// TIA Portal V18 export
TYPE "TM_Pulse_2x24_In_PWM"
   STRUCT
      ERR_PWR : Bool;
      ERR_24V : Bool;
      ERR_LD : Bool;
      Reserved5 : Bool;
      ERR_DQA : Bool;
      ERR_DQB : Bool;
      ERR_OUT_VAL : Bool;
      ERR_SLOT_VAL : Bool;
      Reserved0 : Bool;
      Reserved1 : Bool;
      STS_LD_SLOT : Bool;
      Reserved2 : Bool;
      STS_READY : Bool;
      STS_SW_ENABLE : Bool;
      Reserved3 : Bool;
      Reserved4 : Bool;
      STS_ENABLE : Bool;
      STS_DQA : Bool;
      STS_DQB : Bool;
      STS_DI : Bool;
      STS_DITHER : Bool;
      Reserved6 : Bool;
      Reserved7 : Bool;
      Reserved8 : Bool;
      MEASURE_CURRENT : Int;
      QLMN_LLM : Bool;
      QLMN_HLM : Bool;
      Reserved9 : Bool;
      Reserved10 : Bool;
      Reserved11 : Bool;
      Reserved12 : Bool;
      Reserved13 : Bool;
      Reserved14 : Bool;
      Reserved15 : Byte;
   END_STRUCT;
END_TYPE
